FUNCTION_BLOCK FB_TcAxis_Codesys IMPLEMENTS TMP.itfAxis
VAR_INPUT
END_VAR
VAR_OUTPUT
END_VAR
VAR
END_VAR

{warning 'Agregar implementación de método'}
METHOD AccelerationProfile : itfCommand
VAR_INPUT
	TimeScale	: REAL;
	AccelerationScale	: REAL;
	Offset	: REAL;
	BufferMode	: MC_BUFFER_MODE;
END_VAR
// NETWORK 1
END_METHOD

{warning 'Agregar implementación de propiedad'}
PROPERTY ActualPosition : REAL
GET
// NETWORK 1
END_GET
END_PROPERTY

{warning 'Agregar implementación de propiedad'}
PROPERTY ActualTorque : REAL
GET
// NETWORK 1
END_GET
END_PROPERTY

{warning 'Agregar implementación de propiedad'}
PROPERTY ActualVelocity : REAL
GET
// NETWORK 1
END_GET
END_PROPERTY

{warning 'Agregar implementación de propiedad'}
PROPERTY AxisWarning : BOOL
GET
// NETWORK 1
END_GET
END_PROPERTY

{warning 'Agregar implementación de método'}
METHOD CamIn : itfSynchronizedAxisCommand
VAR_INPUT
	Master	: itfAxis_Tc2_MC2;
	MasterOffset	: REAL;
	SlaveOffset	: REAL;
	MasterScaling	: REAL;
	SlaveScaling	: REAL;
	MasterStartDistance	: REAL;
	MasterSyncPosition	: REAL;
	StartMode	: MC_StartMode;
	MasterValueSource	: MC_Source;
	CamTable	: itfCamTable;
	BufferMode	: MC_BUFFER_MODE;
END_VAR
// NETWORK 1
END_METHOD

{warning 'Agregar implementación de método'}
METHOD CombineAxes : itfSynchronizedAxisCommand
VAR_INPUT
	Master1	: itfAxis_Tc2_MC2;
	Master2	: itfAxis_Tc2_MC2;
	CombineMode	: MC_COMBINE_MODE;
	GearRatioNumeratorM1	: INT;
	GearRatioDenominatorM1	: INT;
	GearRatioNumeratorM2	: INT;
	GearRatioDenominatorM2	: INT;
	MasterValueSourceM1	: MC_SOURCE;
	MasterValueSourceM2	: MC_SOURCE;
	BufferMode	: MC_BUFFER_MODE;
END_VAR
// NETWORK 1
END_METHOD

{warning 'Agregar implementación de propiedad'}
PROPERTY CommunicationReady : BOOL
GET
// NETWORK 1
END_GET
END_PROPERTY

{warning 'Agregar implementación de propiedad'}
PROPERTY Direction : AXIS_DIRECTION
GET
// NETWORK 1
END_GET
END_PROPERTY

{warning 'Agregar implementación de propiedad'}
PROPERTY ErrorId : WORD
GET
// NETWORK 1
END_GET
END_PROPERTY

{warning 'Agregar implementación de método'}
METHOD GearIn : itfSynchronizedAxisCommand
VAR_INPUT
	Master	: itfAxis_Tc2_MC2;
	Ratio	: REAL;
	MasterValueSource	: INT;
	Acceleration	: REAL;
	Deceleration	: REAL;
	Jerk	: REAL;
	BufferMode	: MC_BUFFER_MODE;
END_VAR
// NETWORK 1
END_METHOD

{warning 'Agregar implementación de método'}
METHOD GearInPos : itfSynchronizedAxisCommand
VAR_INPUT
	Master	: itfAxis_Tc2_MC2;
	RatioNumerator	: REAL;
	RatioDenominator	: REAL;
	MasterValueSource	: MC_SOURCE;
	MasterSyncPosition	: REAL;
	SlaveSyncPosition	: REAL;
	SyncMode	: MC_SYNC_MODE;
	MasterStartDistance	: REAL;
	Velocity	: REAL;
	Acceleration	: REAL;
	Deceleration	: REAL;
	Jerk	: REAL;
	BufferMode	: MC_BUFFER_MODE;
END_VAR
// NETWORK 1
END_METHOD

{warning 'Agregar implementación de método'}
METHOD Halt : itfAxisCommand
VAR_INPUT
	Deceleration	: REAL;
	Jerk	: REAL;
	BufferMode	: MC_BUFFER_MODE;
END_VAR
// NETWORK 1
END_METHOD

{warning 'Agregar implementación de método'}
METHOD HaltSuperimposed : itfAxisCommand
VAR_INPUT
	Deceleration	: REAL;
	Jerk	: REAL;
END_VAR
// NETWORK 1
END_METHOD

{warning 'Agregar implementación de método'}
METHOD Home : itfAxisCommand
VAR_INPUT
	Position	: REAL;
	Velocity	: REAL;
	EndVelocity	: REAL;
	Acceleration	: REAL;
	Deceleration	: REAL;
	Jerk	: REAL;
	Direction	: MC_Direction;
	HomingMode	: INT;
	BufferMode	: MC_BUFFER_MODE;
END_VAR
// NETWORK 1
END_METHOD

{warning 'Agregar implementación de propiedad'}
PROPERTY HomeAbsSwitch : BOOL
GET
// NETWORK 1
END_GET
END_PROPERTY

{warning 'Agregar implementación de propiedad'}
PROPERTY IsHomed : BOOL
GET
// NETWORK 1
END_GET
END_PROPERTY

{warning 'Agregar implementación de propiedad'}
PROPERTY LimitSwitchNegative : BOOL
GET
// NETWORK 1
END_GET
END_PROPERTY

{warning 'Agregar implementación de propiedad'}
PROPERTY LimitSwitchPositive : BOOL
GET
// NETWORK 1
END_GET
END_PROPERTY

{warning 'Agregar implementación de propiedad'}
PROPERTY MotionStatus : MOTION_STATUS
GET
// NETWORK 1
END_GET
END_PROPERTY

{warning 'Agregar implementación de método'}
METHOD MoveAbsolute : itfAxisCommand
VAR_INPUT
	Position	: REAL;
	Velocity	: REAL;
	Acceleration	: REAL;
	Deceleration	: REAL;
	Jerk	: REAL;
	Direction	: MC_Direction;
	BufferMode	: MC_BUFFER_MODE;
END_VAR
// NETWORK 1
END_METHOD

{warning 'Agregar implementación de método'}
METHOD MoveAdditive : itfAxisCommand
VAR_INPUT
	Distance	: REAL;
	Velocity	: REAL;
	Acceleration	: REAL;
	Deceleration	: REAL;
	Jerk	: REAL;
	BufferMode	: MC_BUFFER_MODE;
END_VAR
// NETWORK 1
END_METHOD

{warning 'Agregar implementación de método'}
METHOD MoveContinuousAbsolute : itfContinuousAxisCommand
VAR_INPUT
	Position	: REAL;
	EndVelocity	: REAL;
	Velocity	: REAL;
	Acceleration	: REAL;
	Deceleration	: REAL;
	Jerk	: REAL;
	Direction	: MC_DIRECTION;
	BufferMode	: MC_BUFFER_MODE;
END_VAR
// NETWORK 1
END_METHOD

{warning 'Agregar implementación de método'}
METHOD MoveContinuousRelative : itfContinuousAxisCommand
VAR_INPUT
	Distance	: REAL;
	EndVelocity	: REAL;
	Velocity	: REAL;
	Acceleration	: REAL;
	Deceleration	: REAL;
	Jerk	: REAL;
	Direction	: MC_DIRECTION;
	BufferMode	: MC_BUFFER_MODE;
END_VAR
// NETWORK 1
END_METHOD

{warning 'Agregar implementación de método'}
METHOD MoveRelative : itfAxisCommand
VAR_INPUT
	Distance	: REAL;
	Velocity	: REAL;
	Acceleration	: REAL;
	Deceleration	: REAL;
	Jerk	: REAL;
	BufferMode	: MC_BUFFER_MODE;
END_VAR
// NETWORK 1
END_METHOD

{warning 'Agregar implementación de método'}
METHOD MoveSuperimposed : itfAxisCommand
VAR_INPUT
	Distance	: REAL;
	VelocityDiff	: REAL;
	Acceleration	: REAL;
	Deceleration	: REAL;
	Jerk	: REAL;
END_VAR
// NETWORK 1
END_METHOD

{warning 'Agregar implementación de método'}
METHOD MoveVelocity : itfContinuousAxisCommand
VAR_INPUT
	Velocity	: REAL;
	Acceleration	: REAL;
	Deceleration	: REAL;
	Jerk	: REAL;
	Direction	: MC_Direction;
	BufferMode	: MC_BUFFER_MODE;
END_VAR
// NETWORK 1
END_METHOD

{warning 'Agregar implementación de método'}
METHOD PhasingAbsolute : itfSynchronizedAxisCommand
VAR_INPUT
	Master	: itfAxis_Tc2_MC2;
	PhaseShift	: REAL;
	Velocity	: REAL;
	Acceleration	: REAL;
	Deceleration	: REAL;
	Jerk	: REAL;
	BufferMode	: MC_BUFFER_MODE;
END_VAR
// NETWORK 1
END_METHOD

{warning 'Agregar implementación de método'}
METHOD PhasingRelative : itfSynchronizedAxisCommand
VAR_INPUT
	Master	: itfAxis_Tc2_MC2;
	PhaseShift	: REAL;
	Velocity	: REAL;
	Acceleration	: REAL;
	Deceleration	: REAL;
	Jerk	: REAL;
	BufferMode	: MC_BUFFER_MODE;
END_VAR
// NETWORK 1
END_METHOD

{warning 'Agregar implementación de método'}
METHOD PositionProfile : itfCommand
VAR_INPUT
	TimeScale	: REAL;
	PositionScale	: REAL;
	Offset	: REAL;
	BufferMode	: MC_BUFFER_MODE;
END_VAR
// NETWORK 1
END_METHOD

{warning 'Agregar implementación de método'}
METHOD Power : itfCommand
VAR_INPUT
	Enable	: BOOL;
	EnablePositive	: BOOL;
	EnableNegative	: BOOL;
END_VAR
// NETWORK 1
END_METHOD

{warning 'Agregar implementación de propiedad'}
PROPERTY PowerOn : BOOL
GET
// NETWORK 1
END_GET
END_PROPERTY

{warning 'Agregar implementación de método'}
METHOD ReadBoolParameter : MC_Error
VAR_INPUT
	ParameterNumber	: INT;
END_VAR
VAR_OUTPUT
	Value	: BOOL;
END_VAR
// NETWORK 1
END_METHOD

{warning 'Agregar implementación de método'}
METHOD ReadParameter : MC_Error
VAR_INPUT
	ParameterNumber	: INT;
END_VAR
VAR_OUTPUT
	Value	: REAL;
END_VAR
// NETWORK 1
END_METHOD

{warning 'Agregar implementación de propiedad'}
PROPERTY ReadyForPowerOn : BOOL
GET
// NETWORK 1
END_GET
END_PROPERTY

{warning 'Agregar implementación de método'}
METHOD Release : MC_Error
// NETWORK 1
END_METHOD

{warning 'Agregar implementación de método'}
METHOD Reset : itfCommand
// NETWORK 1
END_METHOD

{warning 'Agregar implementación de método'}
METHOD SetOverride : MC_Error
VAR_INPUT
	VelFactor	: REAL;
	AccFactor	: REAL;
	JerkFactor	: REAL;
END_VAR
// NETWORK 1
END_METHOD

{warning 'Agregar implementación de método'}
METHOD SetPosition : itfCommand
VAR_INPUT
	Position	: REAL;
	Relative	: BOOL;
	ExecutionMode	: MC_ExecutionMode;
END_VAR
// NETWORK 1
END_METHOD

{warning 'Agregar implementación de propiedad'}
PROPERTY Simulation : BOOL
GET
// NETWORK 1
END_GET
END_PROPERTY

{warning 'Agregar implementación de propiedad'}
PROPERTY Status : AXIS_STATUS
GET
// NETWORK 1
END_GET
END_PROPERTY

{warning 'Agregar implementación de método'}
METHOD Stop : itfAxisCommand
VAR_INPUT
	Deceleration	: REAL;
	Jerk	: REAL;
END_VAR
// NETWORK 1
END_METHOD

{warning 'Agregar implementación de método'}
METHOD TorqueControl : itfAxisCommand
VAR_INPUT
	Torque	: REAL;
	TorqueRamp	: REAL;
	Velocity	: REAL;
	Acceleration	: REAL;
	Deceleration	: REAL;
	Jerk	: REAL;
	Direction	: MC_DIRECTION;
	BufferMode	: MC_BUFFER_MODE;
END_VAR
// NETWORK 1
END_METHOD

{warning 'Agregar implementación de método'}
METHOD VelocityProfile : itfCommand
VAR_INPUT
	TimeScale	: REAL;
	VelocityScale	: REAL;
	Offset	: REAL;
	BufferMode	: MC_BUFFER_MODE;
END_VAR
// NETWORK 1
END_METHOD

{warning 'Agregar implementación de método'}
METHOD WriteBoolParameter : MC_Error
VAR_INPUT
	ParameterNumber	: INT;
	Value	: BOOL;
END_VAR
// NETWORK 1
END_METHOD

{warning 'Agregar implementación de método'}
METHOD WriteParameter : MC_Error
VAR_INPUT
	ParameterNumber	: INT;
	Value	: REAL;
END_VAR
// NETWORK 1
END_METHOD

END_FUNCTION_BLOCK

(* stored: Version 1.1.0.1, ProductVersion 3.1.4024.12
   POU FB_TcAxis_Codesys: Id {e50bd83f-404e-44dd-b16f-166da0d5a892}, SpecialFunc None
   Method AccelerationProfile: Id {f6b21c16-3707-4aa3-b96c-040e6c2ee5e9}
   Property ActualPosition: Id {ecd6bdfe-f9f4-4082-9637-3eb539377161}
   Get Get: Id {7306c7d7-4dfa-4eb9-9573-4aecae58097c}
   Property ActualTorque: Id {b67fdb3e-329b-4c72-b59c-5758ec537ed8}
   Get Get: Id {fd1f7efd-0c6a-4dd0-a7b0-50ec550870c4}
   Property ActualVelocity: Id {6837ce3d-e7af-4294-bb1f-a4b665ab22b5}
   Get Get: Id {a8f9edfa-63be-4734-8005-39c7b2c3e226}
   Property AxisWarning: Id {6d13089a-3a5e-4cdb-9836-719a7aaccd5c}
   Get Get: Id {f7b9b489-21d2-4da0-9098-75ada6ba0411}
   Method CamIn: Id {3cdfe206-c8bd-4852-96fe-97b082752548}
   Method CombineAxes: Id {4979ae12-7f46-4584-b22c-4d34241d2afe}
   Property CommunicationReady: Id {3e391435-1804-4ea0-9d7c-15e7767d84b4}
   Get Get: Id {61fbf2b1-cd11-4b80-b7d5-23bcb5394b0c}
   Property Direction: Id {47b53d58-0cdd-4bc3-bd0e-b3eb036bbd1f}
   Get Get: Id {ed483b6f-adf8-42f5-b004-0ee38f20fc9b}
   Property ErrorId: Id {7987884e-473c-4375-a624-2a00facbe49c}
   Get Get: Id {c3677ff1-8bca-4074-bb05-856eefe5de10}
   Method GearIn: Id {77138364-5b83-4cf6-938f-556ab88879a0}
   Method GearInPos: Id {98d9bc99-ed23-456e-8e02-1d29d431507e}
   Method Halt: Id {17bd12e5-b884-4250-b10d-ab820cec9cd5}
   Method HaltSuperimposed: Id {e5fc3ee3-395b-4a6b-8f2e-4ec3933e6169}
   Method Home: Id {dbcccf17-d9a7-4c76-993f-cc24da88c577}
   Property HomeAbsSwitch: Id {ade4e613-2a00-4f02-95d4-c9ebeb3f9cdf}
   Get Get: Id {cec00b34-a232-4783-88d0-9947dd67d5cf}
   Property IsHomed: Id {e7acc7dc-26c4-4b18-9268-7f7868d9144b}
   Get Get: Id {5291d9c9-6c48-42fb-9e36-4052017b8e21}
   Property LimitSwitchNegative: Id {6c03c139-23cf-4302-bcc2-8583004e85d2}
   Get Get: Id {00ad368a-004b-46d3-8c40-233f2f490b04}
   Property LimitSwitchPositive: Id {0e32b5ab-8921-45e8-9637-49ccd35da748}
   Get Get: Id {f37bb154-e4e4-45a4-9011-db305b26f1c2}
   Property MotionStatus: Id {544d0e45-824a-43e0-9377-5ec7e991978a}
   Get Get: Id {7260f7c2-bff9-4d6e-9c20-3d2ece5ebcd6}
   Method MoveAbsolute: Id {4b98fd6b-2a2c-4109-b171-3305ea655a1c}
   Method MoveAdditive: Id {dbfab193-37bb-4204-87b0-bc7dd41b8286}
   Method MoveContinuousAbsolute: Id {f0bb6939-ca1c-4127-9b7c-50d846304a7f}
   Method MoveContinuousRelative: Id {33d63ccc-9f1e-4949-b44a-bc7ca4b1e91a}
   Method MoveRelative: Id {4d67e2c3-d058-443b-93d4-40721a832207}
   Method MoveSuperimposed: Id {1a0ecad8-21c6-4856-9357-e8dce720c4fe}
   Method MoveVelocity: Id {eb8c2b0b-48d5-4c6a-842b-bc4ea98f0ec1}
   Method PhasingAbsolute: Id {e774d7c8-f735-4ec2-b020-e0d89355b14d}
   Method PhasingRelative: Id {d7c863d5-3346-4201-9cb5-04caba69de00}
   Method PositionProfile: Id {68ed3cf0-2da0-4d1e-9c15-e9aa9435a9df}
   Method Power: Id {60823f4d-0ee8-488e-982f-9fc0f8bd340a}
   Property PowerOn: Id {94767465-1b48-4e21-854b-a26ee912ba9a}
   Get Get: Id {0e526fbd-037e-4144-a5bb-1b08ea5ae751}
   Method ReadBoolParameter: Id {3c3fb5b3-4f37-4b1c-947f-94333c7487ea}
   Method ReadParameter: Id {43f1a274-d522-4e9b-bb1f-caeb4e5b71e4}
   Property ReadyForPowerOn: Id {ac5118df-a906-4356-81a4-68806e984686}
   Get Get: Id {613e18a4-86e5-485b-95a9-1f76c7700b4d}
   Method Release: Id {d2bd2912-14b5-4c68-a0b2-d94b159b3603}
   Method Reset: Id {dfbbacc1-ad40-4eca-a134-289ee74c689b}
   Method SetOverride: Id {3911bbd1-0357-45c5-95c1-65927fcd6cdf}
   Method SetPosition: Id {8ff2d3c2-fe26-4d9b-9d8d-6dd9a9c2b52f}
   Property Simulation: Id {267bbf4c-6c65-43e8-a98d-3fb57e75a654}
   Get Get: Id {1477ca46-bf82-44ad-b6d8-651b3efe62be}
   Property Status: Id {417e74f3-9857-49fb-95d4-b6c1dc505893}
   Get Get: Id {cfef9609-1673-4d36-9b20-a8b53f7fe5d7}
   Method Stop: Id {8c3ae43a-b34c-41a6-9502-511821ff2659}
   Method TorqueControl: Id {d39d62cf-7a1d-4e6e-bf7b-e9490c438482}
   Method VelocityProfile: Id {f0a1b440-9eef-435d-b92e-ac4119c6c739}
   Method WriteBoolParameter: Id {69b3affa-b15f-47a3-bbfb-83d89e922b7b}
   Method WriteParameter: Id {12ac0cdd-e731-47a2-bb23-33c69d694aa0} *)
